(* IEC 61131-3 sources: AXOpen/src/components.balluff.identification/app/SystemConstants, 2 files *)

(* ---- plc_line_HwIdentifiers.st ---- *)
CONFIGURATION HardwareIDs
    VAR_GLOBAL CONSTANT
        BNIPNT507005Z040_HwID : UINT := UINT#260;
        BNIPNT507005Z040_BIS_M_4XX_045_1_BIS_M_4XX_045_HwID : UINT := UINT#263;
        BNIPNT507005Z040_BNIPNT507005Z040_HwID : UINT := UINT#262;
        BNIPNT507005Z040_BNIPNT507005Z040_BNI_PNT_507_005_Z040_HwID : UINT := UINT#267;
        BNIPNT507005Z040_BNIPNT507005Z040_profinet_HwID : UINT := UINT#257;
        BNIPNT507005Z040_BNIPNT507005Z040_profinet_port_1___M12_HwID : UINT := UINT#258;
        BNIPNT507005Z040_BNIPNT507005Z040_profinet_port_2___M12_HwID : UINT := UINT#259;
        BNIPNT507005Z040_Rack_HwID : UINT := UINT#261;
        BNIPNT507005Z040_Standard_I_O_2_Standard_I_O_HwID : UINT := UINT#266;
        BNIPNT507005Z040_Standard_I_O_3_Standard_I_O_HwID : UINT := UINT#265;
        BNIPNT507005Z040_Standard_I_O_4_Standard_I_O_HwID : UINT := UINT#264;
        PROFINET_IO_System_HwID : UINT := UINT#256;
        plc_line_HwID : UINT := UINT#32;
        plc_line_Rail_0_HwID : UINT := UINT#268;
        plc_line_plc_line_HwID : UINT := UINT#48;
        plc_line_plc_line__plc_line_HwID : UINT := UINT#49;
        plc_line_plc_line_CPU_display_1_HwID : UINT := UINT#54;
        plc_line_plc_line_CPU_exec_unit_1_HwID : UINT := UINT#52;
        plc_line_plc_line_Card_reader_writer_1_HwID : UINT := UINT#51;
        plc_line_plc_line_DP_interface_1_HwID : UINT := UINT#60;
        plc_line_plc_line_LicenseManager_1_HwID : UINT := UINT#42;
        plc_line_plc_line_OPC_UA_1_HwID : UINT := UINT#117;
        plc_line_plc_line_PROFINET_interface_2_HwID : UINT := UINT#72;
        plc_line_plc_line_PROFINET_interface_2_Port_1_HwID : UINT := UINT#73;
        plc_line_plc_line_Virtual_communication_interface_HwID : UINT := UINT#135;
        plc_line_plc_line_plc_line_HwID : UINT := UINT#50;
        plc_line_plc_line_profinet_x1_HwID : UINT := UINT#64;
        plc_line_plc_line_profinet_x1_Port1_HwID : UINT := UINT#65;
        plc_line_plc_line_profinet_x1_Port2_HwID : UINT := UINT#66;

    END_VAR
END_CONFIGURATION

(* ---- plc_line_IoAddresses.st ---- *)
CONFIGURATION IoAddresses
    VAR_GLOBAL
        BNIPNT507005Z040_BIS_M_4XX_045_1_InputAddress_0 AT %IW0: WORD;
        BNIPNT507005Z040_BIS_M_4XX_045_1_InputAddress_1 AT %IW2: WORD;
        BNIPNT507005Z040_BIS_M_4XX_045_1_InputAddress_2 AT %IW4: WORD;
        BNIPNT507005Z040_BIS_M_4XX_045_1_InputAddress_3 AT %IW6: WORD;
        BNIPNT507005Z040_BIS_M_4XX_045_1_InputAddress_4 AT %IW8: WORD;
        BNIPNT507005Z040_BIS_M_4XX_045_1_OutputAddress_0 AT %QW0: WORD;
        BNIPNT507005Z040_BIS_M_4XX_045_1_OutputAddress_1 AT %QW2: WORD;
        BNIPNT507005Z040_BIS_M_4XX_045_1_OutputAddress_2 AT %QW4: WORD;
        BNIPNT507005Z040_BIS_M_4XX_045_1_OutputAddress_3 AT %QW6: WORD;
        BNIPNT507005Z040_BIS_M_4XX_045_1_OutputAddress_4 AT %QW8: WORD;

    END_VAR
END_CONFIGURATION
